PROGRAM P_Demo_FB_BARSunblindTwilightAutomatic
VAR
    fb : FB_BARSunblindTwilightAutomatic;                            // 被演示 FB 实例
    eDataSecurityType_in : E_HVACDataSecurityType ;
    bEnable_in : BOOL := FALSE;
    uiBrightness_in : UINT := 0;
    uiActivateValue_io : UINT := 0;
    uiDeactivateValue_io : UINT := 0;
    uiActivateDelay_io : UINT := 0;
    uiDeactivateDelay_io : UINT := 0;
    uiPositionActiveMode_io : UINT := 0;
    iAngleActiveMode_io : INT := 0;
    stSunblind_out : ST_BARSunblind;
    bActive_out : BOOL;
    uiRemainingTimeActivate_out : UINT;
    uiRemainingTimeDeactivate_out : UINT;
    bError_out : BOOL;
    udiErrorId_out : UDINT;
END_VAR

// ============================================================================
// Tc2_HVAC.FB_BARSunblindTwilightAutomatic 演示程序
// ============================================================================
// 场景：把本 FB 实例化到一个 PLC 程序里，每周期单次调用；按需要把 VAR_INPUT 与
//       VAR_IN_OUT 接到工程信号；VAR_OUTPUT 写入对应监视变量。
// 价值：使用本 FB 比手写状态机 / 控制算法节省大量代码；与 Tc2_HVAC 体系内其它 FB
//       直接对接，命名 / 持久化 / 模式仲裁等约定一致。具体语义见 FB_BARSunblindTwilightAutomatic.md 主文档。
// 验证步骤：
//   1. 右键 PLC 项目下 POUs 文件夹 → Add → Existing Item → 选本 .TcPOU 文件
//   2. 引用 Tc2_HVAC（References → Add library）
//   3. 编译 → 登录 → 运行
//   4. 在线写各 *_in 输入信号触发 FB；在线 monitor *_out 引脚观察状态
// ============================================================================

fb(
    eDataSecurityType := eDataSecurityType_in,
    bEnable := bEnable_in,
    uiBrightness := uiBrightness_in,
    uiActivateValue := uiActivateValue_io,
    uiDeactivateValue := uiDeactivateValue_io,
    uiActivateDelay := uiActivateDelay_io,
    uiDeactivateDelay := uiDeactivateDelay_io,
    uiPositionActiveMode := uiPositionActiveMode_io,
    iAngleActiveMode := iAngleActiveMode_io,
    stSunblind => stSunblind_out,
    bActive => bActive_out,
    uiRemainingTimeActivate => uiRemainingTimeActivate_out,
    uiRemainingTimeDeactivate => uiRemainingTimeDeactivate_out,
    bError => bError_out,
    udiErrorId => udiErrorId_out
);

END_PROGRAM

(* stored: Version 1.1.0.1, ProductVersion 3.1.4024.5
   POU P_Demo_FB_BARSunblindTwilightAutomatic: Id {f71db1a3-447d-5383-a047-32761f68d732}, SpecialFunc None *)
